PROGRAM HMI_Controller
VAR
END_VAR

END_PROGRAM

(* stored: Version 1.1.0.1, ProductVersion 3.1.4022.18
   POU HMI_Controller: Id {521f5e38-1cb7-446b-8876-1aa8d0f3da0a}, SpecialFunc None *)
